# EPICS autosave request: tests/testfiles/cfg/SF_timing_spp_PV.req
$(SYS).DESC
$(SYS)-Code-SP
$(SYS)-DelayInRes-SP
$(SYS)-Freq-SP
